(* IEC 61131-3 sources: Word/plc-course/10-structured-text/labs/starter, 4 files *)

(* ---- 10-1-array-statistics.st ---- *)
(* Lab 10-1: Array statistics - ten cold-store temperature probes.
   Module 10 (Structured Text). STARTER - the declarations are done for you;
   write the logic where it says TODO, then run:
     python3 tools/plctest.py 10-structured-text/labs/starter/10-1-array-statistics.st *)

PROGRAM ArrayStats
  VAR (* interface: the I/O mapping routine copies the ten probe readings in here *)
    Samples  : ARRAY[1..10] OF REAL;  (* probe temperatures, degC. Samples[3] is probe TT-303 *)
    MinValue : REAL;                  (* coldest reading, degC *)
    MaxValue : REAL;                  (* warmest reading, degC *)
    Average  : REAL;                  (* mean of the ten readings, degC *)
    MaxIndex : INT;                   (* probe number (1..10) of the warmest reading *)
  END_VAR
  VAR CONSTANT
    NUM_PROBES : INT := 10;           (* must match the upper bound of Samples *)
  END_VAR
  VAR
    i   : INT;                        (* loop index *)
    Sum : REAL;                       (* running total *)
  END_VAR

  (* TODO: replace these placeholder lines with a FOR loop over Samples that
     finds the minimum, the maximum, the probe number of the maximum and the
     average. Think about what the minimum and maximum should start from. *)
  MinValue := 0.0;
  MaxValue := 0.0;
  Average := 0.0;
  MaxIndex := 0;
END_PROGRAM

CONFIGURATION Config0
  RESOURCE Res0 ON PLC
    TASK MainTask(INTERVAL := T#10ms, PRIORITY := 0);
    PROGRAM Inst0 WITH MainTask : ArrayStats;
  END_RESOURCE
END_CONFIGURATION

(* ---- 10-2-median-filter.st ---- *)
(* Lab 10-2: Median filter for a noisy tank level.
   Module 10 (Structured Text). STARTER - the declarations are done for you;
   write the logic where it says TODO, then run:
     python3 tools/plctest.py 10-structured-text/labs/starter/10-2-median-filter.st *)

PROGRAM MedianFilter
  VAR (* interface *)
    RawLevel      : REAL;   (* noisy level from the radar transmitter, % *)
    SampleTrig    : BOOL;   (* sample clock: each rising edge takes one sample *)
    FilteredLevel : REAL;   (* median of the last five samples, % *)
    Ready         : BOOL;   (* TRUE once five samples have been collected *)
  END_VAR
  VAR (* suggested internal variables - change them if you prefer another design *)
    History    : ARRAY[1..5] OF REAL;  (* samples in arrival order *)
    Sorted     : ARRAY[1..5] OF REAL;  (* working copy to sort *)
    Count      : INT;                  (* samples collected so far, 0..5 *)
    SampleEdge : R_TRIG;               (* rising-edge detector for SampleTrig *)
    i, j       : INT;
    Temp       : REAL;
  END_VAR

  (* TODO:
     1. On each rising edge of SampleTrig, add RawLevel to the history and
        drop the oldest sample.
     2. Set Ready once five samples have been collected.
     3. While not Ready, pass the newest sample through. When Ready, sort a
        copy of the history and output the middle value. *)
  FilteredLevel := 0.0;
  Ready := FALSE;
END_PROGRAM

CONFIGURATION Config0
  RESOURCE Res0 ON PLC
    TASK MainTask(INTERVAL := T#10ms, PRIORITY := 0);
    PROGRAM Inst0 WITH MainTask : MedianFilter;
  END_RESOURCE
END_CONFIGURATION

(* ---- 10-3-strapping-table.st ---- *)
(* Lab 10-3: Tank strapping table - level to volume by piecewise-linear lookup.
   Module 10 (Structured Text). STARTER - the declarations are done for you;
   write the logic where it says TODO, then run:
     python3 tools/plctest.py 10-structured-text/labs/starter/10-3-strapping-table.st *)

PROGRAM StrappingTable
  VAR (* interface *)
    Level      : REAL;   (* measured level, m (already scaled from the 4-20 mA signal) *)
    Volume     : REAL;   (* volume in the tank, m3 *)
    OutOfTable : BOOL;   (* TRUE when Level is below the first or above the last breakpoint *)
    (* Strapping table of a horizontal cylindrical tank, 2.0 m diameter and
       5.0 m long (15.708 m3 when full). The test may load other tables. *)
    LevelBP  : ARRAY[1..9] OF REAL := [0.0, 0.25, 0.5, 0.75, 1.0, 1.25, 1.5, 1.75, 2.0];
    VolumeBP : ARRAY[1..9] OF REAL := [0.0, 1.133, 3.071, 5.380, 7.854, 10.328, 12.637, 14.575, 15.708];
  END_VAR
  VAR (* add your own working variables here *)
    i : INT;
  END_VAR

  (* TODO: clamp outside the table and set OutOfTable; otherwise find the
     segment that contains Level and interpolate between its two ends.
     You may write a FUNCTION for the lookup (see the lesson), or put the
     loop here in the program. *)
  Volume := 0.0;
  OutOfTable := FALSE;
END_PROGRAM

CONFIGURATION Config0
  RESOURCE Res0 ON PLC
    TASK MainTask(INTERVAL := T#10ms, PRIORITY := 0);
    PROGRAM Inst0 WITH MainTask : StrappingTable;
  END_RESOURCE
END_CONFIGURATION

(* ---- 10-4-alarm-message.st ---- *)
(* Lab 10-4: Build an alarm message string for the operator.
   Module 10 (Structured Text). STARTER - the declarations are done for you;
   write the logic where it says TODO, then run:
     python3 tools/plctest.py 10-structured-text/labs/starter/10-4-alarm-message.st *)

PROGRAM AlarmMessage
  VAR (* interface *)
    TagName : STRING := 'TT-104';   (* instrument tag *)
    Units   : STRING := 'degC';     (* engineering units *)
    PV      : REAL;                 (* process value, -3000.0 .. 3000.0 *)
    HiHi    : BOOL;                 (* alarm states from the alarm logic *)
    Hi      : BOOL;
    Lo      : BOOL;
    LoLo    : BOOL;
    BadPV   : BOOL;                 (* signal fault: the value cannot be trusted *)
    Message : STRING;               (* text for the alarm banner, '' when healthy *)
  END_VAR
  VAR (* suggested working variables *)
    Tenths    : INT;      (* PV rounded to whole tenths *)
    ValueText : STRING;   (* PV formatted with one decimal place *)
    StateText : STRING;   (* 'HIGH HIGH', 'HIGH', ... *)
  END_VAR

  (* TODO:
     1. Format PV with one decimal place into ValueText, using REAL_TO_INT,
        integer division, MOD and INT_TO_STRING. Watch the sign.
     2. Build Message with CONCAT, highest priority first:
        BadPV, HiHi, LoLo, Hi, Lo, otherwise ''. *)
  Message := CONCAT(TagName, ' TODO');
END_PROGRAM

CONFIGURATION Config0
  RESOURCE Res0 ON PLC
    TASK MainTask(INTERVAL := T#10ms, PRIORITY := 0);
    PROGRAM Inst0 WITH MainTask : AlarmMessage;
  END_RESOURCE
END_CONFIGURATION
